// TwinCAT 3 PLC project PLC_NoOOP
// ProgramVersion: 3.1.4023.0
// libraries:
//   Tc2_Standard, * (Beckhoff Automation GmbH)
//   Tc2_System, * (Beckhoff Automation GmbH)
//   Tc3_Module, * (Beckhoff Automation GmbH)
// project tree:
//   GVLs/ GVL.TcGVL
//   / PlcTask.TcTTO
//   POUs/ MAIN.TcPOU
// (motion and I/O tree: see PLC project plc)
// real-time tasks:
//   TASK PlcTask: cycle T#10ms, priority 20, ADS port 350
//   TASK PlcTask1: cycle T#10ms, priority 21, ADS port 351

CONFIGURATION PLC_NoOOP
    RESOURCE PLC ON TwinCAT3
        TASK PlcTask(INTERVAL := T#10ms, PRIORITY := 21);
        PROGRAM MAIN WITH PlcTask : MAIN;
    END_RESOURCE
END_CONFIGURATION

// ---- GVLs/GVL.TcGVL
{attribute 'qualified_only'}
VAR_GLOBAL
	EmergencyStopButton				AT%I*	: BOOL;
	StopButton						AT%I*	: BOOL;
	StartButton						AT%I*	: BOOL;
	ProductDetectedSensor			AT%I*	: BOOL;
	ConveyorFullSensor				AT%I*	: BOOL;

	MotorContactor					AT%Q*	: BOOL;
END_VAR

// ---- POUs/MAIN.TcPOU
PROGRAM MAIN
VAR
	ConveyorControl				: BOOL;
	Timeout						: TOF;
END_VAR

// Conveyor control is ok when the ES nor the stop button is pushed
IF NOT GVL.StopButton OR NOT GVL.EmergencyStopButton	THEN
	ConveyorControl	:= FALSE;
	
ELSIF gvl.StartButton	AND gvl.StopButton				THEN
	ConveyorControl	:= TRUE;
	
END_IF

// Minimum time the conveyor keeps on running
Timeout(IN:= ConveyorControl AND gvl.ProductDetectedSensor, PT:=T#5S, Q=> , ET=> );
// Conveyor keeps on running until not full and some extra time
gvl.MotorContactor	:= ConveyorControl AND Timeout.Q AND NOT gvl.ConveyorFullSensor;

END_PROGRAM
